// TIA Portal V17 export
// export: Created 2022-07-20T07:02:35.4084318Z, ExportSetting WithDefaults, DisplayName Totally Integrated Automation Portal, DisplayVersion V17, DisplayName TIA Portal Openness, DisplayVersion V17, DisplayName TIA Portal Version Control Interface, DisplayVersion V17, DisplayName SINAMICS Startdrive Advanced, DisplayVersion V17, DisplayName SINAMICS Startdrive G130, G150, S120, S150, SINAMICS MV, S210, DisplayVersion V17, DisplayName SINAMICS Startdrive G110M, G120, G120C, G120D, G120P, G115D, DisplayVersion V17, DisplayName STEP 7 Professional, DisplayVersion V17, DisplayName STEP 7 Safety, DisplayVersion V17, DisplayName WinCC Advanced, DisplayVersion V17
VAR_GLOBAL   // PLC tag table "ES_IFoilOne"
   DI_2008_0 AT %I2008.0 : Bool;
   DI_2008_1 AT %I2008.1 : Bool;
   DI_2008_2 AT %I2008.2 : Bool;
   DI_2008_3 AT %I2008.3 : Bool;
   DI_2008_4 AT %I2008.4 : Bool;
   DI_2008_5 AT %I2008.5 : Bool;
   DI_2008_6 AT %I2008.6 : Bool;
   DI_2008_7 AT %I2008.7 : Bool;
   DI_2009_0 AT %I2009.0 : Bool;
   DI_2009_1 AT %I2009.1 : Bool;
   DI_2009_2 AT %I2009.2 : Bool;
   DI_2009_3 AT %I2009.3 : Bool;
   DI_2009_4 AT %I2009.4 : Bool;
   DI_2009_5 AT %I2009.5 : Bool;
   DI_2009_6 AT %I2009.6 : Bool;
   DI_2009_7 AT %I2009.7 : Bool;
   DI_2010_0 AT %I2010.0 : Bool;
   DI_2010_1 AT %I2010.1 : Bool;
   DI_2010_2 AT %I2010.2 : Bool;
   DI_2010_3 AT %I2010.3 : Bool;
   DI_2010_4 AT %I2010.4 : Bool;
   DI_2010_5 AT %I2010.5 : Bool;
   DI_2010_6 AT %I2010.6 : Bool;
   DI_2010_7 AT %I2010.7 : Bool;
   DI_2011_0 AT %I2011.0 : Bool;
   DI_2011_1 AT %I2011.1 : Bool;
   DI_2011_2 AT %I2011.2 : Bool;
   DI_2011_3 AT %I2011.3 : Bool;
   DI_2011_4 AT %I2011.4 : Bool;
   DI_2011_5 AT %I2011.5 : Bool;
   DI_2011_6 AT %I2011.6 : Bool;
   DI_2011_7 AT %I2011.7 : Bool;
   DO_2008_0 AT %Q2008.0 : Bool;
   DO_2008_1 AT %Q2008.1 : Bool;
   DO_2008_2 AT %Q2008.2 : Bool;
   DO_2008_3 AT %Q2008.3 : Bool;
   DO_2008_4 AT %Q2008.4 : Bool;
   DO_2008_5 AT %Q2008.5 : Bool;
   DO_2008_6 AT %Q2008.6 : Bool;
   DO_2008_7 AT %Q2008.7 : Bool;
   DO_2009_0 AT %Q2009.0 : Bool;
   DO_2009_1 AT %Q2009.1 : Bool;
   DO_2009_2 AT %Q2009.2 : Bool;
   DO_2009_3 AT %Q2009.3 : Bool;
   DO_2009_4 AT %Q2009.4 : Bool;
   DO_2009_5 AT %Q2009.5 : Bool;
   DO_2009_6 AT %Q2009.6 : Bool;
   DO_2009_7 AT %Q2009.7 : Bool;
   DO_2010_0 AT %Q2010.0 : Bool;
   DO_2010_1 AT %Q2010.1 : Bool;
   DO_2010_2 AT %Q2010.2 : Bool;
   DO_2010_3 AT %Q2010.3 : Bool;
   DO_2010_4 AT %Q2010.4 : Bool;
   DO_2010_5 AT %Q2010.5 : Bool;
   DO_2010_6 AT %Q2010.6 : Bool;
   DO_2010_7 AT %Q2010.7 : Bool;
   DO_2011_0 AT %Q2011.0 : Bool;
   DO_2011_1 AT %Q2011.1 : Bool;
   DO_2011_2 AT %Q2011.2 : Bool;
   DO_2011_3 AT %Q2011.3 : Bool;
   DO_2011_4 AT %Q2011.4 : Bool;
   DO_2011_5 AT %Q2011.5 : Bool;
   DO_2011_6 AT %Q2011.6 : Bool;
   DO_2011_7 AT %Q2011.7 : Bool;
   AI_2000_0 AT %IW2000 : Int;
   AI_2000_1 AT %IW2002 : Int;
   AO_2000_0 AT %QW2000 : Int;
   AO_2000_1 AT %QW2002 : Int;
   AI_2000_2 AT %IW2004 : Int;
   AI_2000_3 AT %IW2006 : Int;
END_VAR
